PROGRAM RunMotor
VAR
END_VAR

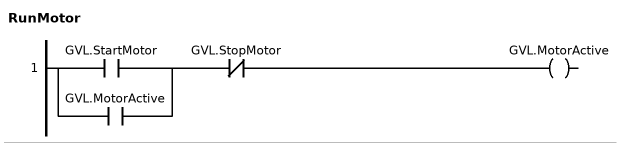
// NETWORK 1
GVL.MotorActive := (GVL.StartMotor OR GVL.MotorActive) AND NOT GVL.StopMotor;

END_PROGRAM

(* stored: Version 1.1.0.1, ProductVersion 3.1.4024.12
   POU RunMotor: Id {b63b43fa-8e36-408e-865a-bb277ea9fe78}, SpecialFunc None *)
